{attribute addProperty BoxType "EJ7411-0000-0018"}
{attribute addProperty Id "FB_PositionAT %I*FB_Position_BA8AA9F03240DRV_StatuswordAT %I*DRV_Statusword_53CBCECC1620DRV_Following_error_actual_valueAT %I*DRV_Following_error_actual_value_F54335363240DRV_ControlwordAT %Q*DRV_Controlword_417617681620DRV_Target_positionAT %Q*DRV_Target_position_41334FAA3240WcStateAT %I*WcState_98A4DF7520.250InfoDataAT %I*InfoData_81099714160200"}
{attribute addProperty CRC "4078408466"}
{attribute addProperty SizeInBites "290"}
{attribute addProperty SizeInBytes "36.25"}
TYPE EJ7411_675FBD05 :
STRUCT
	{attribute addProperty Name "FB_Position"}
	FB_Position : FB_Position_BA8AA9F0;
	{attribute addProperty Name "DRV_Statusword"}
	DRV_Statusword : DRV_Statusword_53CBCECC;
	{attribute addProperty Name "DRV_Following_error_actual_value"}
	DRV_Following_error_actual_value : DRV_Following_error_actual_value_F5433536;
	{attribute addProperty Name "DRV_Controlword"}
	DRV_Controlword : DRV_Controlword_41761768;
	{attribute addProperty Name "DRV_Target_position"}
	DRV_Target_position : DRV_Target_position_41334FAA;
	{attribute addProperty Name "WcState"}
	WcState : WcState_98A4DF75;
	{attribute addProperty Name "InfoData"}
	InfoData : InfoData_81099714;
END_STRUCT
END_TYPE

(* stored: Version 1.2.0.0, ProductVersion 3.1.4024.9
   DUT EJ7411_675FBD05: Id {297b402d-193a-4947-841a-b5544fc006d4} *)
